FUNCTION_BLOCK FB_CalcLREALMock EXTENDS FB_FallibleMock IMPLEMENTS I_CalcLREAL
VAR
    fResult : LREAL;
END_VAR


METHOD Calculate : LREAL

Calculate := fResult;
END_METHOD


METHOD SetResult
VAR_INPUT
    fResult : LREAL;
END_VAR

THIS^.fResult := fResult;
END_METHOD

END_FUNCTION_BLOCK

(* stored: Version 1.1.0.1
   POU FB_CalcLREALMock: Id {bd34b3e8-fd89-4e8a-b12d-4532c72a5f8a}, SpecialFunc None
   Method Calculate: Id {8d2db5d4-517a-48a1-b360-7ddccbfcc9d8}
   Method SetResult: Id {83f2d6c6-eaa9-4112-bf0b-9f218db5e2c1} *)
